INTERFACE I_ExampleInterface EXTENDS __SYSTEM.IQueryInterface

END_INTERFACE

(* stored: Version 1.1.0.1, ProductVersion 3.1.4024.11
   Itf I_ExampleInterface: Id {ac253b9b-dbad-4f27-a366-b96e21128b21} *)
